TYPE ST_System_HES_Parameter :
STRUCT
	AutoQuittierung			: BOOL;
END_STRUCT
END_TYPE

(* stored: Version 1.1.0.1, ProductVersion 3.1.4024.9
   DUT ST_System_HES_Parameter: Id {f27c723f-1afc-4724-9b70-26356093eda8} *)
